FUNCTION_BLOCK FB_MqttClient
VAR_INPUT
END_VAR
VAR_OUTPUT
END_VAR
VAR
    fbMqttClient : FB_IotMqttClient;
    sTopicToPublish: STRING(255) := 'Temperature'; 	// MQTT topic for temperature
    sMessageToPublish: STRING(255); 				// Message buffer
    tmrSendMessageInterval: TON := (PT := T#1S); 	// Interval timer for publishing
    ai_RoomTemperature: INT := 1; 					// Room temperature from thermocouple
	is_init : BOOL := FALSE;
END_VAR

fbMqttClient.sClientId:= 'Publishing PLC';
fbMqttClient.sHostName:= '158.180.44.197';
fbMqttClient.nHostPort:= 1883;
fbMqttClient.sTopicPrefix:= 'aut/apt-get rekt/'; 
fbMqttClient.sUserName:= 'bobm';
fbMqttClient.sUserPassword:= 'letmein';

fbMqttClient.Execute(bConnect := TRUE);

//METH_Publish('$$groupname', 'apt-get rekt');
//METH_Publish('names', 'Erdogan - Holzmann - Jolfai');
//METH_Publish('bEnable', bool_to_string(IFC_HW.bEnable));
METH_Publish('bEnable/$$unit', 'BOOL');

METHOD METH_Publish : BOOL
VAR_INPUT
	sTopicToPublish : STRING;
	sMessageToPublish : STRING;
END_VAR
IF fbMqttClient.bConnected THEN
    tmrSendMessageInterval(IN := TRUE);
    IF tmrSendMessageInterval.Q THEN
        tmrSendMessageInterval(IN := FALSE);
        //sMessageToPublish := REAL_TO_STRING(ai_RoomTemperature / 10.0);

        fbMqttClient.Publish(
            sTopic := sTopicToPublish,
            pPayload := ADR(sMessageToPublish),
            nPayloadSize := LEN(sMessageToPublish) + 1,
            eQoS := TcIotMqttQos.AtMostOnceDelivery,
            bRetain := TRUE,
            bQueue := TRUE
        );
    END_IF
END_IF
END_METHOD

END_FUNCTION_BLOCK

(* stored: Version 1.1.0.1, ProductVersion 3.1.4024.15
   POU FB_MqttClient: Id {3e717b62-5220-4ec3-aa52-f14d56865976}, SpecialFunc None
   Method METH_Publish: Id {01defe36-a556-483c-9626-a78d51726ba9} *)
